// TIA Portal V20 export
DATA_BLOCK "CS_Drive_PL"   // DB13, Motion_DB
// stored: InstanceOfName TO_SynchronousAxis, OfSystemLibElement TO_SynchronousAxis, OfSystemLibVersion 7.0
TO_SynchronousAxis   // technology object, version 7.0
// stored: Connection Interface Actor, InputAddress 9256, OutputAddress 9256
// stored: Connection Interface Sensor[1], InputAddress 9256, OutputAddress 9256, SensorIndexInActorTelegram 1
// stored: Connection Interface Sensor[2], SensorIndexInActorTelegram 1, PathToDBMember EncoderTel81.Tel81.Sensor_1
// stored: Connection Interface Torque, InputAddress 10352, OutputAddress 10352
// stored: SetPointCoupling Ref CS_Virtual_Axis, Type TO_PositioningAxis
   // // inherited from TO_PositioningAxis
   // // inherited from TO_SpeedAxis
   // // inherited from TO_Axis
   // // inherited from TO_Object
   // VAR
   //    Actor : TO_Struct_Actor;
   //    LoadGear : TO_Struct_LoadGear;
   // END_VAR
   // VAR
   //    Sensor : Array[1..4] of TO_Struct_Sensor;
   //    Mechanics : TO_Struct_Mechanics;
   //    PositionControl : TO_Struct_PositionControl;
   //    DynamicAxisModel : TO_Struct_DynamicAxisModel;
   //    FollowingError : TO_Struct_FollowingError;
   //    PositioningMonitoring : TO_Struct_PositioningMonitoring;
   //    StandstillSignal : TO_Struct_StandstillSignal;
   // END_VAR
   // VAR
   //    StatusSynchronizedMotion { ExternalWritable := 'False'; S7_SetPoint := 'True'} : TO_Struct_StatusSynchronizedMotion;
   // END_VAR
BEGIN
   Actor.InverseDirection := true;
   Actor.DataAdaption := 1;
   Actor.Interface.AddressIn.RID := 16#208072a;
   Actor.Interface.AddressIn.AREA := 16#81;
   Actor.Interface.AddressIn.OFFSET := 9256;
   Actor.Interface.AddressOut.RID := 16#208072b;
   Actor.Interface.AddressOut.AREA := 16#82;
   Actor.Interface.AddressOut.OFFSET := 9256;
   Actor.Interface.TorqueDataAddressIn.RID := 16#2080742;
   Actor.Interface.TorqueDataAddressOut.RID := 16#2080743;
   Actor.DriveParameter.ReferenceSpeed := 6000.0;
   Actor.DriveParameter.MaxSpeed := 6000.0;
   Actor.DriveParameter.ReferenceTorque := 47.04;
   LoadGear.Numerator := 6843;
   LoadGear.Denominator := 100;
   Sensor[1]."Type" := 2;
   Sensor[2]."Type" := 1;
   Sensor[1].InverseDirection := true;
   Sensor[2].System := 0;
   Sensor[2].MountingMode := 1;
   Sensor[1].DataAdaption := 1;
   Sensor[1].Interface.AddressIn.RID := 16#208072a;
   Sensor[2].Interface.AddressIn.RID := 16#208070e;
   Sensor[1].Interface.AddressIn.AREA := 16#81;
   Sensor[1].Interface.AddressIn.OFFSET := 9256;
   Sensor[1].Interface.AddressOut.RID := 16#208072b;
   Sensor[2].Interface.AddressOut.RID := 16#208070f;
   Sensor[1].Interface.AddressOut.AREA := 16#82;
   Sensor[1].Interface.AddressOut.OFFSET := 9256;
   Sensor[2].Parameter.Resolution := 1.0;
   Sensor[2].Parameter.FineResolutionXist1 := 0;
   Sensor[1..2].Parameter.FineResolutionXist2 := 0;
   Sensor[1].Parameter.DeterminableRevolutions := 4096;
   Mechanics.LeadScrew := 1256.0;
   PositionControl.Kv := 1.5;
   PositionControl.EnableDSC := true;
   DynamicAxisModel.VelocityTimeConstant := 0.004;
   FollowingError.MinValue := 20.0;
   FollowingError.MinVelocity := 20.0;
   PositioningMonitoring.Window := 5.0;
   StandstillSignal.VelocityThreshold := 10.0;
   Sensor[2].Type := 1;
   _Actor.Interface.Telegram := 105;
   _Actor.DataAdaptionOffline := True;
   _Sensor[1].Interface.Telegram := 105;
   _Sensor[1].DataAdaptionOffline := True;
   _Sensor[2].Interface.Telegram := 81;
END_DATA_BLOCK
